% RSLogix 500 project Pump_Protection.RSS, saved by version 8.30.00.16 %
PROJECT "UNTITLED"    % processor: Bul.1763 MicroLogix 1100 Series B %

PROGRAM FILES
  LAD 2 "MAIN"  5 rungs
  LAD 3 "DIGITAL IO"  5 rungs
  LAD 4 "CONTROLS"  7 rungs

DATA FILES
  O0 OUTPUT  4 elements
  I1 INPUT  6 elements
  S2 STATUS  66 elements
  B3 BINARY  1 elements
  T4 TIMER  2 elements
  C5 COUNTER  1 elements
  R6 CONTROL  1 elements
  N7 INTEGER  1 elements
  F8 FLOAT  1 elements

LADDER 2 "MAIN"
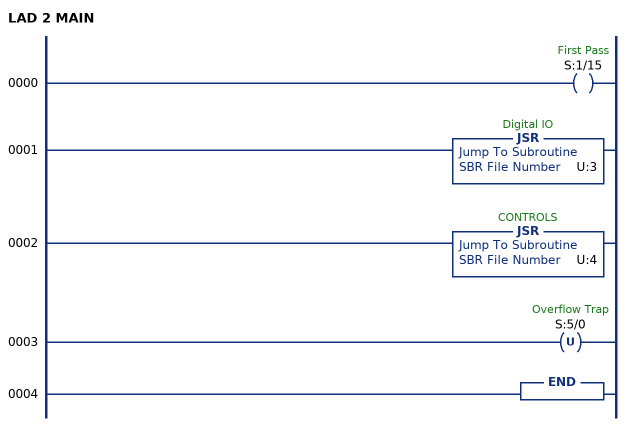
% Rung: 0 %
SOR OTE S:1/15 EOR
%   S:1/15  "First Pass" %
% Rung: 1 %
SOR JSR U:3 EOR
%   U:3  "Digital IO" %
% Rung: 2 %
SOR JSR U:4 EOR
%   U:4  "CONTROLS" %
% Rung: 3 %
SOR OTU S:5/0 EOR
%   S:5/0  "Overflow Trap" %
% Rung: 4 %
SOR END EOR

LADDER 3 "DIGITAL IO"
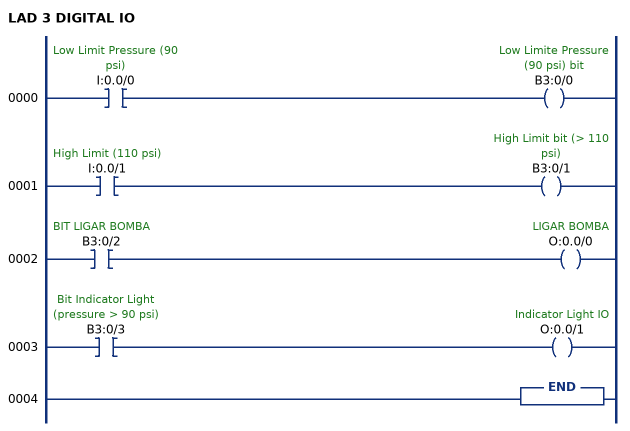
% Rung: 0 %
SOR XIC I:0.0/0 OTE B3:0/0 EOR
%   I:0.0/0  "Low Limit Pressure (90 psi)" %
%   B3:0/0  "Low Limite Pressure (90 psi) bit" %
% Rung: 1 %
SOR XIC I:0.0/1 OTE B3:0/1 EOR
%   I:0.0/1  "High Limit (110 psi)" %
%   B3:0/1  "High Limit bit (> 110 psi)" %
% Rung: 2 %
SOR XIC B3:0/2 OTE O:0.0/0 EOR
%   B3:0/2  "BIT LIGAR BOMBA" %
%   O:0.0/0  "LIGAR BOMBA" %
% Rung: 3 %
SOR XIC B3:0/3 OTE O:0.0/1 EOR
%   B3:0/3  "Bit Indicator Light (pressure > 90 psi)" %
%   O:0.0/1  "Indicator Light IO" %
% Rung: 4 %
SOR END EOR

LADDER 4 "CONTROLS"
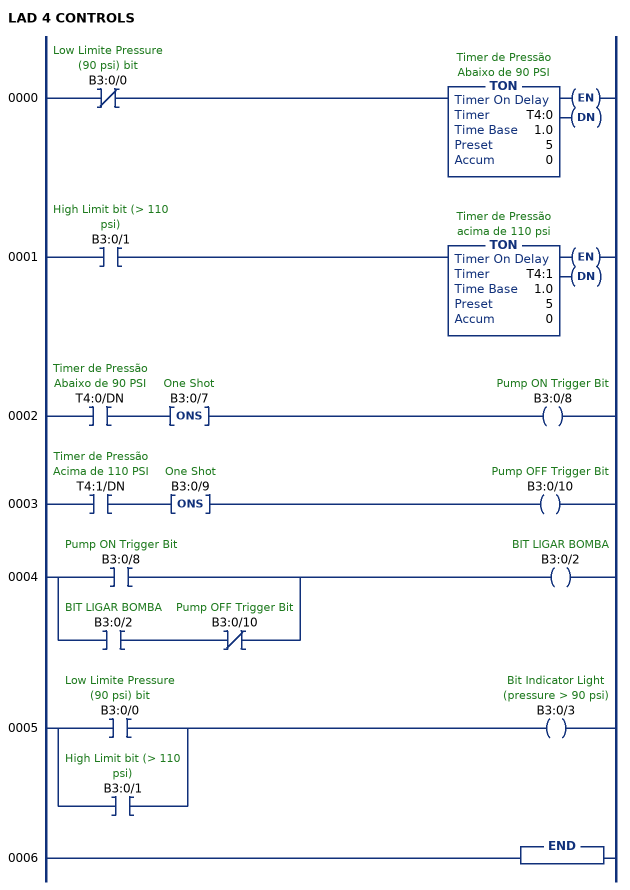
% Rung: 0 %
SOR XIO B3:0/0 TON T4:0 1.0 5 0 EOR
%   B3:0/0  "Low Limite Pressure (90 psi) bit" %
%   T4:0  "Timer de Pressão Abaixo de 90 PSI" %
% Rung: 1 %
SOR XIC B3:0/1 TON T4:1 1.0 5 0 EOR
%   B3:0/1  "High Limit bit (> 110 psi)" %
%   T4:1  "Timer de Pressão acima de 110 psi" %
% Rung: 2 %
SOR XIC T4:0/DN ONS B3:0/7 OTE B3:0/8 EOR
%   T4:0/DN  "Timer de Pressão Abaixo de 90 PSI" %
%   B3:0/7  "One Shot" %
%   B3:0/8  "Pump ON Trigger Bit" %
% Rung: 3 %
SOR XIC T4:1/DN ONS B3:0/9 OTE B3:0/10 EOR
%   T4:1/DN  "Timer de Pressão Acima de 110 PSI" %
%   B3:0/9  "One Shot" %
%   B3:0/10  "Pump OFF Trigger Bit" %
% Rung: 4 %
SOR BST XIC B3:0/8 NXB XIC B3:0/2 XIO B3:0/10 BND OTE B3:0/2 EOR
%   B3:0/8  "Pump ON Trigger Bit" %
%   B3:0/2  "BIT LIGAR BOMBA" %
%   B3:0/10  "Pump OFF Trigger Bit" %
% Rung: 5 %
SOR BST XIC B3:0/0 NXB XIC B3:0/1 BND OTE B3:0/3 EOR
%   B3:0/0  "Low Limite Pressure (90 psi) bit" %
%   B3:0/1  "High Limit bit (> 110 psi)" %
%   B3:0/3  "Bit Indicator Light (pressure > 90 psi)" %
% Rung: 6 %
SOR END EOR

OTHER DOCUMENTED ADDRESSES
  B3:0/4  "BOTAO DE INICIAR SISTEMA"
  B3:0/5  "One Shot"
  T4:0/TT  "Timer de Pressão abaixo de 90 PSI"
  T4:1/TT  "Começando a contar o tempo com pressão acima de 110 PSI. Devemos desligar a bomba de pressão."

DATA TABLE (non-zero values as saved)
DATA B3
% B3:0 % 0X0004
DATA T4
% .PRE .ACC %
% T4:0 % 5 0
% T4:1 % 5 0
